// TIA Portal V16 export
// export: Created 2021-11-12T13:31:10.4174816Z, ExportSetting WithDefaults, DisplayName Totally Integrated Automation Portal, DisplayVersion V16 Update 3, DisplayName TIA Portal Version Control Interface, DisplayVersion V16 Update 2, DisplayName TIA Portal Openness, DisplayVersion V16 Update 3, DisplayName SINAMICS Startdrive Advanced, DisplayVersion V16 Update 5, DisplayName SINAMICS Startdrive G130, G150, S120, S150, SINAMICS MV, S210, DisplayVersion V16 Update 5, DisplayName SINAMICS Startdrive G110M, G120, G120C, G120D, G120P, G115D, DisplayVersion V16 Update 5, DisplayName STEP 7 Professional, DisplayVersion V16 Update 3, DisplayName STEP 7 Safety, DisplayVersion V16, DisplayName WinCC UA Professional, DisplayVersion V16 Update 3
DATA_BLOCK "Sfty_Status"   // DB7, F_DB
{ S7_Optimized_Access := 'TRUE'; DB_Accessible_From_OPC_UA := 'FALSE' }
VERSION : 0.1
// stored: AutoNumber true, DBAccessibleFromOPCUA false
   VAR
      EStopZone100 : "UDT_Safety";   // Safety zone 100 - emergency stop ok
      EStopZone200 : "UDT_Safety";   // Safety zone 200 - emergency stop ok
      EStopZone300 : "UDT_Safety";   // Safety zone 300 - emergency stop ok
      EStopZone400 : "UDT_Safety";   // Safety zone 400 - emergency stop ok
      FenceZone101 : "UDT_Safety";   // Safety zone 101 - fence ok
      FenceZone102 : "UDT_Safety";   // Safety zone 102 - fence ok
      FenceZone103 : "UDT_Safety";   // Safety zone 103 - fence ok
      FenceZone104 : "UDT_Safety";   // Safety zone 104 - fence ok
      FenceZone105 : "UDT_Safety";   // Safety zone 105 - fence ok
      KAS1_ES : "UDT_Safety";   // Estop from saw machine KAS1
      KAS2_ES : "UDT_Safety";   // Estop from saw machine KAS1
      BSN1_2_ES : "UDT_Safety";   // Estop from owen BSN1 / BSN2
      SCH1_ES : "UDT_Safety";   // Estop from press SCH1
      BSN3_ES : "UDT_Safety";   // Estop from owen BSN3
      BSN4_5_ES : "UDT_Safety";   // Estop from owen BSN4 / BSN5
      THM1_ES : "UDT_Safety";   // Estop from blasting machine THM1
      THM2_ES : "UDT_Safety";   // Estop from blasting machine THM2
      "1R1-RC01_ES" : "UDT_Safety";   // Estop from robot 1R1-RC01
      "1R2-RC01_ES" : "UDT_Safety";   // Estop from robot 1R2-RC01
      "1R3-RC01_ES" : "UDT_Safety";   // Estop from robot 1R3-RC01
      "1R5-RC01_ES" : "UDT_Safety";   // Estop from robot 1R5-RC01
      "1R6-RC01_ES" : "UDT_Safety";   // Estop from robot 1R6-RC01
      "2R1-RC01_ES" : "UDT_Safety";   // Estop from robot 2R1-RC01
      "2R2-RC01_ES" : "UDT_Safety";   // Estop from robot 2R2-RC01
      "000UH11-SF01_12_ES" : "UDT_Safety";   // Estop button central panel
      "000UH10-SF01_12_ES" : "UDT_Safety";   // Estop button central pult
      "100UH11-SF01_12_ES" : "UDT_Safety";   // Estop button control panel 1 - HMI
      "100UH12-SF01_12_ES" : "UDT_Safety";   // Estop button control panel 2 - HMI
      "100UH13-SF01_12_ES" : "UDT_Safety";   // Estop button control panel 3 - HMI
      "100UF01-SF01_12_ES" : "UDT_Safety";   // Estop button control panel 4
      "200UH11-SF01_12_ES" : "UDT_Safety";   // Estop button control panel 1 - HMI
      "200UF01-SF01_12_ES" : "UDT_Safety";   // Estop button control panel 4
      "210UF01-SF01_12_ES" : "UDT_Safety";   // Estop button control panel conveyor 210
      "220UF01-SF01_12_ES" : "UDT_Safety";   // Estop button control panel conveyor 220
      "230UF01-SF01_12_ES" : "UDT_Safety";   // Estop button control panel conveyor 230
      "300UH11-SF01_12_ES" : "UDT_Safety";   // Estop button control panel 1 - HMI
      "310UH31-SF01_12_ES" : "UDT_Safety";   // Estop button control panel 1
      "330UF01-SF01_12_ES" : "UDT_Safety";   // Estop button control panel conveyor 330
      "400UH11-SF01_12_ES" : "UDT_Safety";   // Estop button control panel 1 - HMI
      "400UH31-SF01_12_ES" : "UDT_Safety";   // Estop button control panel 1
      "410UH31-SF01_12_ES" : "UDT_Safety";   // Estop button control panel 2
      "420UH31-SF01_12_ES" : "UDT_Safety";   // Estop button control panel 3
      "100RU01-QQ01_ES" : "UDT_Safety";   // Estop button gate 100RU01-QQ1
      "100RU01-QQ02_ES" : "UDT_Safety";   // Estop button gate 100RU01-QQ2
      "100RU01-QQ03_ES" : "UDT_Safety";   // Estop button gate 100RU01-QQ3
      "100RU01-QQ04_ES" : "UDT_Safety";   // Estop button gate 100RU01-QQ4
      "100RU01-QQ05_ES" : "UDT_Safety";   // Estop button gate 100RU01-QQ5
      "100RU01-QQ06_ES" : "UDT_Safety";   // Estop button gate 100RU01-QQ6
      "100RU01-QQ07_ES" : "UDT_Safety";   // Estop button gate 100RU01-QQ7
      "100RU01-QQ08_ES" : "UDT_Safety";   // Estop button gate 100RU01-QQ8
      "200RU01-QQ01_ES" : "UDT_Safety";   // Estop button gate 200RU01-QQ1
      "200RU01-QQ02_ES" : "UDT_Safety";   // Estop button gate 200RU01-QQ2
      "200RU01-QQ03_ES" : "UDT_Safety";   // Estop button gate 200RU01-QQ3
      "200RU01-QQ04_ES" : "UDT_Safety";   // Estop button gate 200RU01-QQ4
      "200RU01-QQ05_ES" : "UDT_Safety";   // Estop button gate 200RU01-QQ5
      "100RU01-QQ01_Lock" : "UDT_Safety";   // Estop gate 100RU01-QQ1 close&lock
      "100RU01-QQ02_Lock" : "UDT_Safety";   // Estop gate 100RU01-QQ2 close&lock
      "100RU01-QQ03_Lock" : "UDT_Safety";   // Estop gate 100RU01-QQ3 close&lock
      "100RU01-QQ04_Lock" : "UDT_Safety";   // Estop gate 100RU01-QQ4 close&lock
      "100RU01-QQ05_Lock" : "UDT_Safety";   // Estop gate 100RU01-QQ5 close&lock
      "100RU01-QQ06_Lock" : "UDT_Safety";   // Estop gate 100RU01-QQ6 close&lock
      "100RU01-QQ07_Lock" : "UDT_Safety";   // Estop gate 100RU01-QQ7 close&lock
      "100RU01-QQ08_Lock" : "UDT_Safety";   // Estop gate 100RU01-QQ8 close&lock
      "200RU01-QQ01_Lock" : "UDT_Safety";   // Estop gate 200RU01-QQ1 close&lock
      "200RU01-QQ02_Lock" : "UDT_Safety";   // Estop gate 200RU01-QQ2 close&lock
      "200RU01-QQ03_Lock" : "UDT_Safety";   // Estop gate 200RU01-QQ3 close&lock
      "200RU01-QQ04_Lock" : "UDT_Safety";   // Estop gate 200RU01-QQ4 close&lock
      "200RU01-QQ05_Lock" : "UDT_Safety";   // Estop gate 200RU01-QQ5 close&lock
      "100RU01-BG01_4_Fence" : "UDT_Safety";   // Estop fence 1
      "100RU01-BG02_4_Fence" : "UDT_Safety";   // Estop fence 2
      "200RU01-BG01_4 _Fence" : "UDT_Safety";   // Estop tunel to press - sensor
      "100UR01-KG01R_2_Fence" : "UDT_Safety";   // Estop Light barrier input to KAS1
      "100UR01-KG02R_2_Fence" : "UDT_Safety";   // Estop Light barrier input to KAS2
      "100UH01-KF51_A1" : "UDT_Safety";   // Safety relay estop KAS1/KAS2
      "400UH01-KF51_A1" : "UDT_Safety";   // Safety relay estop THM1
      "100UH01-KF52_A1" : "UDT_Safety";   // Safety relay auto stop KAS1
      "100UH01-KF53_A1" : "UDT_Safety";   // Safety relay auto stop KAS2
      "CRS_BSN1/2_Fault" : "UDT_Safety";   // Profisafe communication fault - CRS -> BSN1/2
      CRS_SCH1_Fault : "UDT_Safety";   // Profisafe communication fault - CRS -> SCH1
      CRS_BSN3_Fault : "UDT_Safety";   // Profisafe communication fault - CRS -> BSN3
      "CRS_BSN4/5_Fault" : "UDT_Safety";   // Profisafe communication fault - CRS -> BSN4/5
      "BSN1/2_CRS_Fault" : "UDT_Safety";   // Profisafe communication fault - BSN1/2 - > CRS
      SCH1_CRS_Fault : "UDT_Safety";   // Profisafe communication fault - SCH1 - > CRS
      BSN3_CRS_Fault : "UDT_Safety";   // Profisafe communication fault - BSN3 - > CRS
      "BSN4/5_CRS_Fault" : "UDT_Safety";   // Profisafe communication fault - BSN4/5 - > CRS
      "1R1-RC01_Module" : "UDT_Safety";   // Safety modul fault - 1R1-RC01
      "1R2-RC01_Module" : "UDT_Safety";   // Safety modul fault - 1R2-RC01
      "1R3_1R4-RC01_Module" : "UDT_Safety";   // Safety modul fault - 1R3_1R4-RC01
      "1R5-RC01_Module" : "UDT_Safety";   // Safety modul fault - 1R5-RC01
      "1R6-RC01_Module" : "UDT_Safety";   // Safety modul fault - 1R6-RC01
      "2R1-RC01_Module" : "UDT_Safety";   // Safety modul fault - 2R1-RC01
      "2R2-RC01_Module" : "UDT_Safety";   // Safety modul fault - 2R2-RC01
      "000UH01-KF31_Module" : "UDT_Safety";   // Safety modul fault - 100UH11-KF31
      "000UH01-KF32_Module" : "UDT_Safety";   // Safety modul fault - 000UH01-KF32
      "000UH01-KF33_Module" : "UDT_Safety";   // Safety modul fault - 000UH01-KF33
      "000UH01-KF41_Module" : "UDT_Safety";   // Safety modul fault - 000UH01-KF41
      "000UH11-KF31_Module" : "UDT_Safety";   // Safety modul fault - 000UH11-KF31
      "000UH11-KF32_Module" : "UDT_Safety";   // Safety modul fault - 000UH11-KF32
      "100UH11-KF31_Module" : "UDT_Safety";   // Safety modul fault - 100UH11-KF31
      "100UH12-KF31_Module" : "UDT_Safety";   // Safety modul fault - 100UH12-KF31
      "100UH13-KF31_Module" : "UDT_Safety";   // Safety modul fault - 100UH13-KF31
      "100UH13-KF32_Module" : "UDT_Safety";   // Safety modul fault - 100UH13-KF32
      "200UH11-KF31_Module" : "UDT_Safety";   // Safety modul fault - 200UH11-KF31
      "300UH11-KF31_Module" : "UDT_Safety";   // Safety modul fault - 300UH11-KF31
      "310UH31-KF31_Module" : "UDT_Safety";   // Safety modul fault - 310UH31-KF31
      "400UH11-KF31_Module" : "UDT_Safety";   // Safety modul fault - 400UH11-KF31
      "400UH31-KF31_Module" : "UDT_Safety";   // Safety modul fault - 400UH31-KF31
      "410UH31-KF31_Module" : "UDT_Safety";   // Safety modul fault - 410UH31-KF31
      "420UH31-KF31_Module" : "UDT_Safety";   // Safety modul fault - 420UH31-KF31
      "100+RU01-KF01_Module" : "UDT_Safety";   // Safety door module fault - 100+RU01-KF01
      "100+RU01-KF02_Module" : "UDT_Safety";   // Safety door module fault - 100+RU01-KF02
      "100+RU01-KF03_Module" : "UDT_Safety";   // Safety door module fault - 100+RU01-KF03
      "200+RU01-KF02_Module" : "UDT_Safety";   // Safety door module fault - 200+RU01-KF02
      "200+RU01-KF03_Module" : "UDT_Safety";   // Safety door module fault - 200+RU01-KF03
      "200+RU01-KF04_Module" : "UDT_Safety";   // Safety door module fault - 200+RU01-KF04
      "110+UC12-TA01_Module" : "UDT_Safety";   // Inverter safety module fault - 110+UC12-TA01
      "120+UC12-TA01_Module" : "UDT_Safety";   // Inverter safety module fault - 120+UC12-TA01
      "210+UC12-TA01_Module" : "UDT_Safety";   // Inverter safety module fault - 210+UC12-TA01
      "220+UC12-TA01_Module" : "UDT_Safety";   // Inverter safety module fault - 220+UC12-TA01
      "230+UC12-TA01_Module" : "UDT_Safety";   // Inverter safety module fault - 230+UC12-TA01
      "230+UC12-TA02_Module" : "UDT_Safety";   // Inverter safety module fault - 230+UC12-TA02
      "320+UC21-TA01_Module" : "UDT_Safety";   // Inverter safety module fault - 320+UC21-TA01
      "330+UC21-TA01_Module" : "UDT_Safety";   // Inverter safety module fault - 330+UC21-TA01
      "330+UC21-TA02_Module" : "UDT_Safety";   // Inverter safety module fault - 330+UC21-TA02
      "330+UC21-TA03_Module" : "UDT_Safety";   // Inverter safety module fault - 330+UC21-TA03
      "430+UC21-TA01_Module" : "UDT_Safety";   // Inverter safety module fault - 430+UC21-TA01
      "440+UC21-TA01_Module" : "UDT_Safety";   // Inverter safety module fault - 440+UC21-TA01
      "450+UC21-TA01_Module" : "UDT_Safety";   // Inverter safety module fault - 450+UC21-TA01
      "450+UC21-TA02_Module" : "UDT_Safety";   // Inverter safety module fault - 450+UC21-TA02
      "450+UC21-TA03_Module" : "UDT_Safety";   // Inverter safety module fault - 450+UC21-TA03
      "450+UC21-TA04_Module" : "UDT_Safety";   // Inverter safety module fault - 450+UC21-TA04
      "460+UC21-TA01_Module" : "UDT_Safety";   // Inverter safety module fault - 460+UC21-TA01
      "460+UC21-TA02_Module" : "UDT_Safety";   // Inverter safety module fault - 460+UC21-TA02
      "460+UC21-TA03_Module" : "UDT_Safety";   // Inverter safety module fault - 460+UC21-TA03
      "460+UC21-TA04_Module" : "UDT_Safety";   // Inverter safety module fault - 460+UC21-TA04
   END_VAR
BEGIN
END_DATA_BLOCK
